{attribute 'qualified_only'}
VAR_GLOBAL
	bAroLuzOn: BOOL;
	bAroLuzOff: BOOL;
END_VAR

(* stored: Version 1.1.0.1, ProductVersion 3.1.4024.16
   GVL GVL_ILUMINACION: Id {1e393bf1-bf50-424e-b13e-5a641ea4a0ff} *)
